Fanuc TP program (LS listing): test_1.ls

/PROG  TEST_1
/ATTR
OWNER		= MNEDITOR;
COMMENT		= "";
PROG_SIZE	= 222;
CREATE		= DATE 18-11-16  TIME 15:35:44;
MODIFIED	= DATE 18-11-16  TIME 15:44:30;
FILE_NAME	= ;
VERSION		= 0;
LINE_COUNT	= 6;
MEMORY_SIZE	= 570;
PROTECT		= READ_WRITE;
TCD:  STACK_SIZE	= 0,
      TASK_PRIORITY	= 50,
      TIME_SLICE	= 0,
      BUSY_LAMP_OFF	= 0,
      ABORT_REQUEST	= 0,
      PAUSE_REQUEST	= 0;
DEFAULT_GROUP	= 1,*,*,*,*;
CONTROL_CODE	= 00000000 00000000;
/MN
   1:  UFRAME_NUM=1 ;
   2:  UTOOL_NUM=5 ;
   3:   ;
   4:  PR[1,3:HOME]=(-100)    ;
   5:J PR[10:V_PAL1] 100% CNT50 Tool_Offset,PR[1:HOME]    ;
   6:L PR[10:V_PAL1] 100mm/sec FINE    ;
/POS
/END
